(* IEC 61131-3 sources: DTDFEvaluation/02 persistent storage - SauvegardeEx recordings (example)/home/steam/Schreibtisch/OpenPLC_v3/webserver/st_files, 3 files *)

(* ---- 0-38966.st ---- *)
PROGRAM program0
  VAR
    PB1 AT %MW0.0 : INT;
    PB2 AT %MW0.1 : INT;
    PB3 AT %MW0.2 : INT;
    PB4 AT %MW0.3 : INT;
  END_VAR

  IF PB1<1 THEN
      WHILE PB2 < 8000 DO
          PB2 := PB2 + 1;
          PB3 := PB3 + 10;
          PB4 := PB4 + 20;
      END_WHILE;
  END_IF;
END_PROGRAM

CONFIGURATION Config0

  RESOURCE Res0 ON PLC
    TASK task0(INTERVAL := T#55ms,PRIORITY := 0);
    PROGRAM instance0 WITH task0 : program0;
  END_RESOURCE
END_CONFIGURATION

(* ---- 2-38966.st ---- *)
PROGRAM program0
  VAR
    PB1 AT %MW0.0 : INT;
    PB2 AT %MW0.1 : INT;
    PB3 AT %MW0.2 : INT;
    PB4 AT %MW0.3 : INT;
    PB5 AT %MW0.4 : INT;
    PB6 AT %IX0.5 : INT;
  END_VAR

  PB2 := 0;
  IF TRUE THEN
      WHILE PB2 < 8000 DO
          PB2 := PB2 + 1;
          PB3 := PB3 + 10;
          PB4 := PB4 + 20;
          PB5 := PB5 + 21;
      END_WHILE;
  END_IF;

END_PROGRAM

CONFIGURATION Config0

  RESOURCE Res0 ON PLC
    TASK task0(INTERVAL := T#5s0ms,PRIORITY := 0);
    PROGRAM instance0 WITH task0 : program0;
  END_RESOURCE
END_CONFIGURATION

(* ---- 38966.st ---- *)
PROGRAM program0
  VAR
    PB1 AT %MW0.0 : INT;
    PB2 AT %MW0.1 : INT;
    PB3 AT %MW0.2 : INT;
    PB4 AT %MW0.3 : INT;
    PB5 AT %MW0.4 : INT;
  END_VAR

  IF PB1<1 THEN
      WHILE PB2 < 8000 DO
          PB2 := PB2 + 1;
          PB3 := PB3 + 10;
          PB4 := PB4 + 20;
          PB5 := PB5 + 21;
      END_WHILE;
      PB2 := 0;
      PB3 := 0;
      PB4 := 0;
      PB5 := 0;
  END_IF;

END_PROGRAM

CONFIGURATION Config0

  RESOURCE Res0 ON PLC
    TASK task0(INTERVAL := T#5s0ms,PRIORITY := 0);
    PROGRAM instance0 WITH task0 : program0;
  END_RESOURCE
END_CONFIGURATION
